FUNCTION_BLOCK FB_ExampleDeviceSM
VAR_INPUT
	i_xMoveStarted	:	BOOL; //Connect to moving flag
	i_xMoveDone	:	BOOL; //Connect to move done flag
	i_xBeamReady	:	BOOL; //Connect to transitioneer
	i_xStopDone	:	BOOL; //Connect to MC_Stop.Done
END_VAR
VAR_OUTPUT
	q_xStartMove	:	BOOL; //Connect to MC_Absolute.Execute
	q_xStop			:	BOOL; //Connect to MC_Stop.Execute
	q_rTargetPosition	:	REAL; //Connect to MC_Absolute.Position
	q_stRequiredBeamParametersID	:	UDINT;
	q_stRequiredBeamParameters	:	ST_BeamParams; //Connect to BeamParameterTransitionManager
END_VAR
VAR_IN_OUT
	stDevice	:	ST_Device;
END_VAR
VAR
	nTargetState	:	INT;
	
	xNewReq	:	BOOL; //Set true when new target request present
	
END_VAR

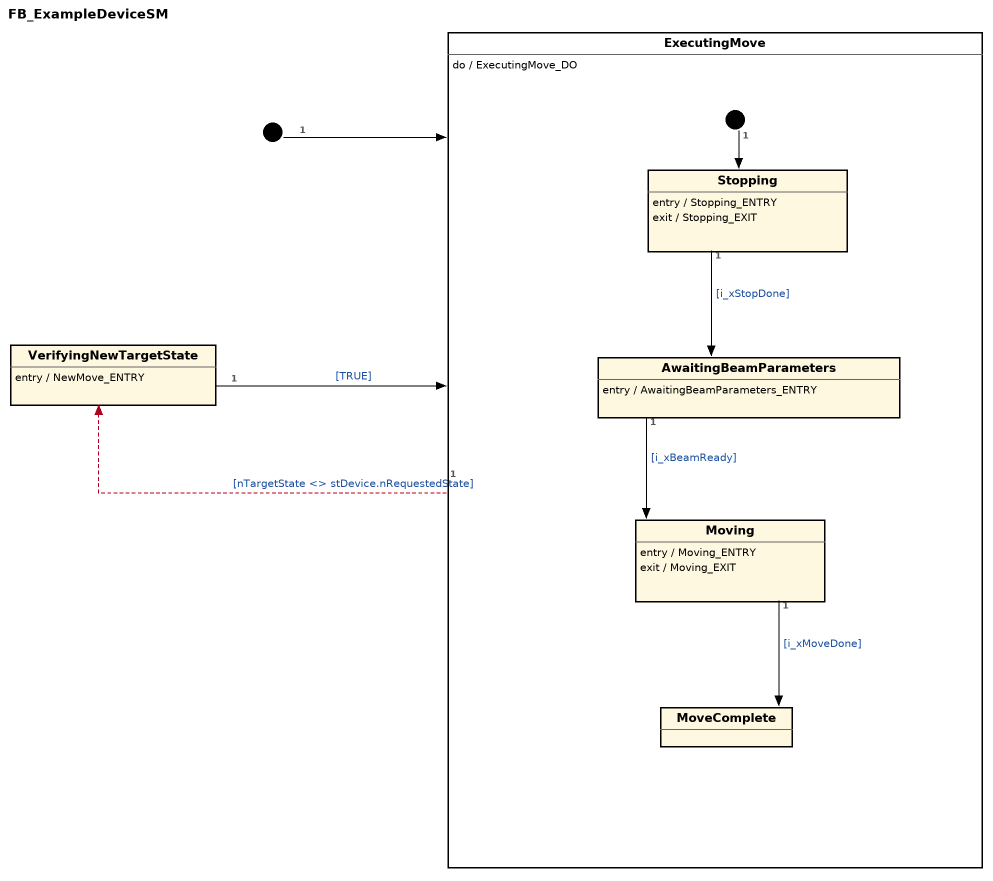
STATECHART FB_ExampleDeviceSM  // abortable
    START StartState1
    COMPOSITE STATE ExecutingMove
        do / ExecutingMove_DO
        START StartState2
        STATE Stopping
            entry / Stopping_ENTRY
            exit / Stopping_EXIT
        STATE AwaitingBeamParameters
            entry / AwaitingBeamParameters_ENTRY
        STATE Moving
            entry / Moving_ENTRY
            exit / Moving_EXIT
        STATE MoveComplete
        StartState2 -> Stopping  // priority 1, on completion
        Stopping -> AwaitingBeamParameters [i_xStopDone] // priority 1, rising edge
        AwaitingBeamParameters -> Moving [i_xBeamReady] // priority 1, rising edge
        Moving -> MoveComplete [i_xMoveDone] // priority 1, rising edge
    END_STATE
    STATE VerifyingNewTargetState
        entry / NewMove_ENTRY
    StartState1 -> ExecutingMove  // priority 1, on completion
    ExecutingMove -> VerifyingNewTargetState [nTargetState <> stDevice.nRequestedState] // priority 1, exception, rising edge
    VerifyingNewTargetState -> ExecutingMove [TRUE] // priority 1
END_STATECHART

ACTION AwaitingBeamParameters_ENTRY:
q_stRequiredBeamParameters := stDevice.astStates[nTargetState].stReqBeamParam;
q_stRequiredBeamParametersID := stDevice.astStates[nTargetState].nStateRef;
END_ACTION

ACTION ExecutingMove_DO:

END_ACTION

ACTION Moving_ENTRY:
q_xStartMove := TRUE;
q_rTargetPosition := stDevice.astStates[nTargetState].rPosition;
END_ACTION

ACTION Moving_EXIT:
q_xStartMove := FALSE;
END_ACTION

ACTION NewMove_ENTRY:

IF stDevice.nRequestedState <= PMPS_GVL.cnMaxStateArrayLen AND
	stDevice.nRequestedState >= 1 THEN
	nTargetState := stDevice.nRequestedState;
END_IF
END_ACTION

ACTION Stopping_ENTRY:
q_xStop	:= TRUE;
END_ACTION

ACTION Stopping_EXIT:
q_xStop := FALSE;
END_ACTION

END_FUNCTION_BLOCK

(* stored: Version 1.1.0.1, ProductVersion 3.1.4022.18
   POU FB_ExampleDeviceSM: Id {2af5974b-b277-059d-24ec-a85477882535}, SpecialFunc None
   Action AwaitingBeamParameters_ENTRY: Id {81e16e47-29b0-0a9a-3d20-fdfeadefa08e}
   Action ExecutingMove_DO: Id {508791e6-c057-0365-16c1-c3b87fb536bf}
   Action Moving_ENTRY: Id {36aa9be1-0e05-0c9b-14a1-9c4f7124e34a}
   Action Moving_EXIT: Id {871ca4d0-de02-04c5-2494-a255e9aa5989}
   Action NewMove_ENTRY: Id {f1754a41-bd83-096a-3203-436ddbae5403}
   Action Stopping_ENTRY: Id {cde0afac-cd3e-0fdf-32ef-6b08364c4df8}
   Action Stopping_EXIT: Id {f1d7f949-a24a-04cd-2456-5a672755c5dd} *)
